Fanuc KAREL source: kt00126.KL

PROGRAM KT00126
%STACKSIZE=65535
%PRIORITY=65535
%NOLOCKGROUP
VAR
OUT : REAL
-- UNRESOLVED DECLARATIONS (source type spelling not recovered)
-- H1 : ARRAY[2] OF TYPE_0x0017 (type_u16=0x2017)
-- Y2 : ARRAY[2] OF TYPE_0x0018 (type_u16=0x2018)
BEGIN
-- UNRESOLVED_PC line 8 opcodes [2E 22 9D 33 B4] marker_code=0
Y2[1]=3
-- UNRESOLVED_PC line 10 opcodes [22 9D 33 B3 22 9D 33 B1 64 29 64 29 6C 23] marker_code=38
END KT00126
